Fanuc KAREL source: KD00007.KL

PROGRAM KD00007
%NOLOCKGROUP
%SHADOWVARS
VAR
  I: INTEGER
  J: INTEGER
  B: BOOLEAN
  R: REAL
  S: STRING[80]
BEGIN
  I = 1
END KD00007
